{attribute 'qualified_only'}
VAR_GLOBAL
	


//	msgArry: ARRAY[1..gHMIDataConst.gNumberOfMessagesScreen] OF typeNewMsg;
//	msgArryStyle: ARRAY[1..gHMIDataConst.gNumberOfMessagesScreen] OF typeNewMsgStyle;
//	msgHeader:typeNewMsgHeader;
	
	
	//new implementation
	//S1_msg :structEventViewMsg;
	
	//nulls do not apply, have to assign to FB
	msgArrynull: ARRAY[1..gHMIDataConst.gNumberOfMessagesScreen] OF typeNewMsg;
	msgArryStylenull: ARRAY[1..gHMIDataConst.gNumberOfMessagesScreen] OF typeNewMsgStyle;
	msgWasChangednull:BOOL;
	
END_VAR

(* stored: Version 1.1.0.1, ProductVersion 3.1.4024.12
   GVL gMsgView: Id {c98a8eb5-ce00-4b7a-bc77-80f3bc5f447e} *)
